// TIA Portal project "Project8" (V15.1)

(* hardware
DEVICE "S7-1200 station_1"  S7-1200 Station
   slot 0: "Rack_0"  S7-1200 Rack  Rack  V1.0
   slot 1: "PLC_1"  CPU 1214C DC/DC/Rly  6ES7 214-1HG40-0XB0  V4.2
*)

// ===== PLC "PLC_1"  CPU 1214C DC/DC/Rly =====

VAR_GLOBAL   // PLC tag table "Default tag table"
   "Tag_1" AT %Q0.0 : Bool;
   "Tag_2" AT %Q0.2 : Bool;
   "Tag_3" AT %Q0.3 : Bool;
   "Tag_4" AT %Q0.1 : Bool;
   "Tag_5" AT %Q0.4 : Bool;
END_VAR

VAR_GLOBAL   // PLC tag table "Tag table_1"
   "toggle buton" AT %I0.0 : Bool;
   "mem0" AT %M0.1 : Bool;
   "mem1" AT %M0.2 : Bool;
   "mem2" AT %M0.3 : Bool;
   "mem3" AT %M0.4 : Bool;
   "cikis" AT %Q0.5 : Bool;
END_VAR

ORGANIZATION_BLOCK "Main"   // OB1, LAD, ProgramCycle
TITLE = "Main Program Sweep (Cycle)"
{ S7_Optimized_Access := 'TRUE' }
VERSION : 0.1
   VAR_INPUT
      Initial_Call : Bool;   // Initial call of this OB
      Remanence : Bool;   // =True, if remanent data are available
   END_VAR
BEGIN

REGION Network 1
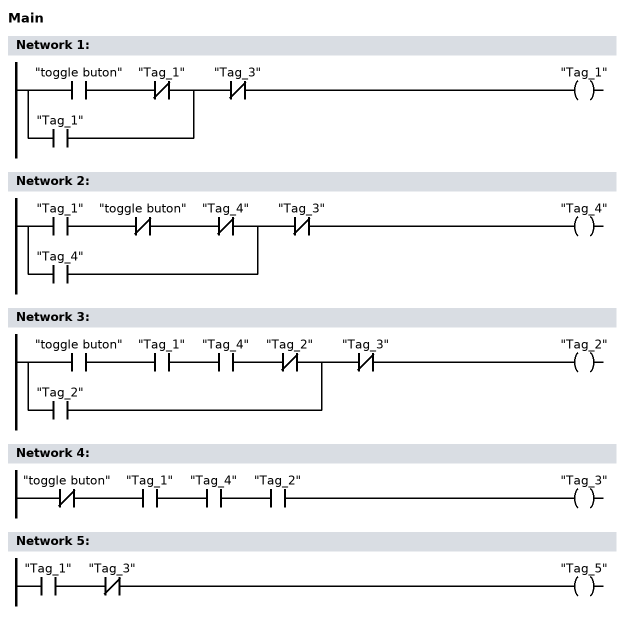
   RUNG wire#powerrail
      Contact( "toggle buton" )
      I_Contact( "Tag_1" )
      wire#w1
      I_Contact( "Tag_3" )
      Coil( "Tag_1" )
   END_RUNG
   RUNG wire#powerrail
      Contact( "Tag_1" )
   END_RUNG wire#w1
   // the same network as SCL:
   "Tag_1" := (("toggle buton" AND NOT "Tag_1") OR "Tag_1") AND NOT "Tag_3";
END_REGION

REGION Network 2
   RUNG wire#powerrail
      Contact( "Tag_1" )
      I_Contact( "toggle buton" )
      I_Contact( "Tag_4" )
      wire#w1
      I_Contact( "Tag_3" )
      Coil( "Tag_4" )
   END_RUNG
   RUNG wire#powerrail
      Contact( "Tag_4" )
   END_RUNG wire#w1
   // the same network as SCL:
   "Tag_4" := (("Tag_1" AND NOT "toggle buton" AND NOT "Tag_4") OR "Tag_4") AND NOT "Tag_3";
END_REGION

REGION Network 3
   RUNG wire#powerrail
      Contact( "toggle buton" )
      Contact( "Tag_1" )
      Contact( "Tag_4" )
      I_Contact( "Tag_2" )
      wire#w1
      I_Contact( "Tag_3" )
      Coil( "Tag_2" )
   END_RUNG
   RUNG wire#powerrail
      Contact( "Tag_2" )
   END_RUNG wire#w1
   // the same network as SCL:
   "Tag_2" := (("toggle buton" AND "Tag_1" AND "Tag_4" AND NOT "Tag_2") OR "Tag_2") AND NOT "Tag_3";
END_REGION

REGION Network 4
   RUNG wire#powerrail
      I_Contact( "toggle buton" )
      Contact( "Tag_1" )
      Contact( "Tag_4" )
      Contact( "Tag_2" )
      Coil( "Tag_3" )
   END_RUNG
   // the same network as SCL:
   "Tag_3" := NOT "toggle buton" AND "Tag_1" AND "Tag_4" AND "Tag_2";
END_REGION

REGION Network 5
   RUNG wire#powerrail
      Contact( "Tag_1" )
      I_Contact( "Tag_3" )
      Coil( "Tag_5" )
   END_RUNG
   // the same network as SCL:
   "Tag_5" := "Tag_1" AND NOT "Tag_3";
END_REGION
END_ORGANIZATION_BLOCK